TYPE CM_Sensor_PAR :
STRUCT
END_STRUCT
END_TYPE

(* stored: Version 1.1.0.1, ProductVersion 3.1.4024.12
   DUT CM_Sensor_PAR: Id {912aa722-8625-49fb-8edb-fe88e61cb0b9} *)
